FUNCTION "CCDB-PLC Factory Call_Devices" : Void
{ S7_Optimized_Access := 'TRUE' }
VERSION : 0.1
   VAR_TEMP
      "false" : Bool;
      "true" : Bool;
   END_VAR


BEGIN
	#false:=0;
	#true := 1;

	"LNS-ISrc-01:Vac-TMPC-1"(    EPICStoPLC_DB:=“EPICStoPLC”,
	                             EPICStoPLC_Offset:=20,
	                             PLCtoEPICS_DB:=“PLCtoEPICS”,
	                             PLCtoEPICS_Offset:=100,
	                             "NominalSpeedSt|OnSt.DI”:=“LNS-LEBT-010:Vac-VEPT-02100:NormalOperation.DI”,
	                             "HardwareError.DI”:=“LNS-LEBT-010:Vac-VEPT-02100:Error.DI”,
	                             "Start.DO”:=“LNS-LEBT-010:Vac-VEPT-02100:START.DO”
							);
########## INSTALLATION_SLOT PLC->EPICS status ##########

record(bi, INSTALLATION_SLOT:ManMode) {
	field(SCAN, "I/O Intr")
	field(DTYP, "S7plc")
	field(INP, "@$(PLCNAME)/88 T=WORD B=0")
}
record(bi, INSTALLATION_SLOT:Closed) {
	field(SCAN, "I/O Intr")
	field(DTYP, "S7plc")
	field(INP, "@$(PLCNAME)/88 T=WORD B=1")
}
record(bi, INSTALLATION_SLOT:Open) {
	field(SCAN, "I/O Intr")
	field(DTYP, "S7plc")
	field(INP, "@$(PLCNAME)/88 T=WORD B=2")
}
record(bi, INSTALLATION_SLOT:LocalMode) {
	field(SCAN, "I/O Intr")
	field(DTYP, "S7plc")
	field(INP, "@$(PLCNAME)/88 T=WORD B=3")
}
record(bi, INSTALLATION_SLOT:ForcedMode) {
	field(SCAN, "I/O Intr")
	field(DTYP, "S7plc")
	field(INP, "@$(PLCNAME)/88 T=WORD B=4")
}
record(bi, INSTALLATION_SLOT:BlockedClosedMode) {
	field(SCAN, "I/O Intr")
	field(DTYP, "S7plc")
	field(INP, "@$(PLCNAME)/88 T=WORD B=5")
}
record(bi, INSTALLATION_SLOT:OpenOutput) {
	field(SCAN, "I/O Intr")
	field(DTYP, "S7plc")
	field(INP, "@$(PLCNAME)/88 T=WORD B=7")
}




record(ai, INSTALLATION_SLOT:InRegister2) {
	field(SCAN, "I/O Intr")
	field(DTYP, "S7plc")
	field(INP, "@$(PLCNAME)/90 T=WORD")
}

record(ai, INSTALLATION_SLOT:InRegister3) {
	field(SCAN, "I/O Intr")
	field(DTYP, "S7plc")
	field(INP, "@$(PLCNAME)/92 T=WORD")
}

record(ai, INSTALLATION_SLOT:InRegister4) {
	field(SCAN, "I/O Intr")
	field(DTYP, "S7plc")
	field(INP, "@$(PLCNAME)/94 T=WORD")
}

record(ai, INSTALLATION_SLOT:InRegister5) {
	field(SCAN, "I/O Intr")
	field(DTYP, "S7plc")
	field(INP, "@$(PLCNAME)/96 T=WORD")
}

record(ai, INSTALLATION_SLOT:InRegister6) {
	field(SCAN, "I/O Intr")
	field(DTYP, "S7plc")
	field(INP, "@$(PLCNAME)/98 T=WORD")
}

record(ai, INSTALLATION_SLOT:InRegister7) {
	field(SCAN, "I/O Intr")
	field(DTYP, "S7plc")
	field(INP, "@$(PLCNAME)/100 T=WORD")
}
####################

########## INSTALLATION_SLOT EPICS->PLC commands ##########

record(bo, INSTALLATION_SLOT:AutoCmd) {
  field(DTYP, "asynUInt32Digital")
  field(OUT,  "@asynMask($(PLCNAME)write, 18, 0x0001, 100)")
}
record(bo, INSTALLATION_SLOT:ManCmd) {
  field(DTYP, "asynUInt32Digital")
  field(OUT,  "@asynMask($(PLCNAME)write, 18, 0x0002, 100)")
}
record(bo, INSTALLATION_SLOT:ManCloseCmd) {
  field(DTYP, "asynUInt32Digital")
  field(OUT,  "@asynMask($(PLCNAME)write, 18, 0x0004, 100)")
}
record(bo, INSTALLATION_SLOT:ManOpenCmd) {
  field(DTYP, "asynUInt32Digital")
  field(OUT,  "@asynMask($(PLCNAME)write, 18, 0x0008, 100)")
}
record(bo, INSTALLATION_SLOT:RemoteCmd) {
  field(DTYP, "asynUInt32Digital")
  field(OUT,  "@asynMask($(PLCNAME)write, 18, 0x0010, 100)")
}
record(bo, INSTALLATION_SLOT:IntlkBypassCmd) {
  field(DTYP, "asynUInt32Digital")
  field(OUT,  "@asynMask($(PLCNAME)write, 18, 0x0020, 100)")
}
record(bo, INSTALLATION_SLOT:BlockClosedCmd) {
  field(DTYP, "asynUInt32Digital")
  field(OUT,  "@asynMask($(PLCNAME)write, 18, 0x0040, 100)")
}
record(bo, INSTALLATION_SLOT:ResetCmd) {
  field(DTYP, "asynUInt32Digital")
  field(OUT,  "@asynMask($(PLCNAME)write, 18, 0x0080, 100)")
}

####################
END_FUNCTION
